FUNCTION_BLOCK FB_Gaszaehler
VAR_INPUT
	Telegramm	: ARRAY[1..cMBUS_MaxTelegrams] OF ST_MBus_Data2;

END_VAR
VAR_IN_OUT
	Zustand		: ST_GZ_Zustand;
END_VAR
VAR
END_VAR
VAR // added by the converter: edge detectors and wires of the graphical bodies
    _w1, _w2, _w3 : ANY;
END_VAR

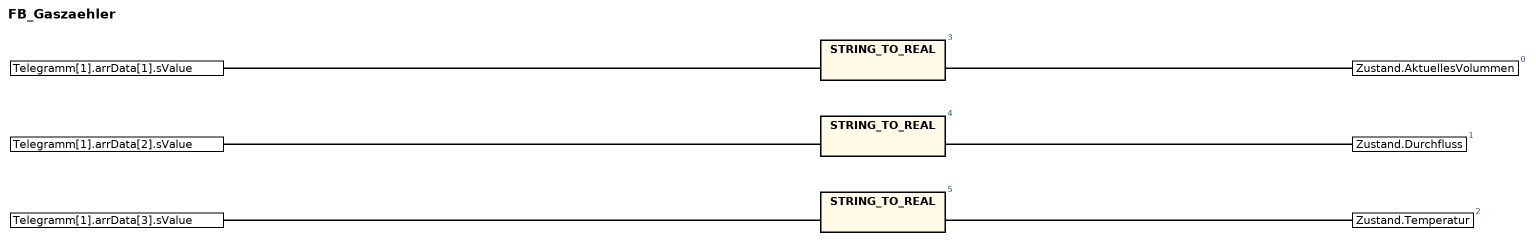
Zustand.AktuellesVolummen := _w1;
Zustand.Durchfluss := _w2;
Zustand.Temperatur := _w3;
_w1 := STRING_TO_REAL(Telegramm[1].arrData[1].sValue);
_w2 := STRING_TO_REAL(Telegramm[1].arrData[2].sValue);
_w3 := STRING_TO_REAL(Telegramm[1].arrData[3].sValue);

END_FUNCTION_BLOCK

(* stored: Version 1.1.0.1, ProductVersion 3.1.4024.9
   POU FB_Gaszaehler: Id {daa49fb7-1b7b-484a-862e-01b03caec40b}, SpecialFunc None *)
